TYPE csp_case_transport_status_enum :
(
	CSP_CASE_TRANSPORT_STATUS_NOT_INITIALIZED 							:=  0,
	CSP_CASE_TRANSPORT_STATUS_DISABLED 									:=  10,
	CSP_CASE_TRANSPORT_STATUS_ENABLE_REQUEST 							:=  20,
	CSP_CASE_TRANSPORT_STATUS_ENABLING 									:=  30,
	CSP_CASE_TRANSPORT_STATUS_ENABLED 									:=  40,
	CSP_CASE_TRANSPORT_STATUS_CHANGE_OVER_MODE							:=  45,
	CSP_CASE_TRANSPORT_STATUS_HOME_REQUEST								:=  50,
	CSP_CASE_TRANSPORT_STATUS_HOMING									:=  60,
	CSP_CASE_TRANSPORT_STATUS_HOME_DONE									:=  70,
	CSP_CASE_TRANSPORT_STATUS_CALCULATING_SLAVE_POSITION				:=  90,
	CSP_CASE_TRANSPORT_STATUS_CALCULATING_MASTER_POSITION				:=  91,
	CSP_CASE_TRANSPORT_STATUS_WAITING_SLAVE_ENGAGE						:= 100,
	CSP_CASE_TRANSPORT_STATUS_WAITING_MASTER_ENGAGE						:= 101,
	CSP_CASE_TRANSPORT_STATUS_PHASE_REQUEST								:= 140,
	CSP_CASE_TRANSPORT_STATUS_PHASING									:= 150,
	CSP_CASE_TRANSPORT_STATUS_PHASED									:= 160,
	CSP_CASE_TRANSPORT_STATUS_CAM_ENGAGED_REQ							:= 170,
	CSP_CASE_TRANSPORT_STATUS_AXIS_ENGAGE_VERIFY						:= 180,
	CSP_CASE_TRANSPORT_STATUS_CAM_ENGAGED								:= 190,
	CSP_CASE_TRANSPORT_STATUS_CAM_TABLE_READ							:= 195,
	CSP_CASE_TRANSPORT_STATUS_CALCULATE_SLAVE_POSITION_REQUEST			:= 196,
	CSP_CASE_TRANSPORT_STATUS_READY										:= 197,
	CSP_CASE_TRANSPORT_STATUS_RUNNING									:= 200,
	CSP_CASE_TRANSPORT_STATUS_MOVING									:= 205,
	CSP_CASE_TRANSPORT_STATUS_DISENGAGE_REQUEST							:= 210,
	CSP_CASE_TRANSPORT_STATUS_DISENGAGING								:= 211,	
	CSP_CASE_TRANSPORT_STATUS_STOP_REQUEST 								:= 500,
	CSP_CASE_TRANSPORT_STATUS_DISABLE_REQUEST 							:= 530,
	CSP_CASE_TRANSPORT_STATUS_DISABLING 								:= 540,
	
	CSP_CASE_TRANSPORT_STATUS_RECOVERY_CAM_ENGAGED_REQ					:= 305,
	CSP_CASE_TRANSPORT_STATUS_DISENGAGE_REJECT							:= 300,
	CSP_CASE_TRANSPORT_STATUS_REJECT_ABS_STEP_1							:= 301,
	CSP_CASE_TRANSPORT_STATUS_REJECT_ABS_STEP_2							:= 302,
	CSP_CASE_TRANSPORT_STATUS_REJECT_ABS_STEP_3							:= 303,
	CSP_CASE_TRANSPORT_STATUS_REJECT_ABS_STEP_4							:= 304	
	
) := CSP_CASE_TRANSPORT_STATUS_NOT_INITIALIZED;
END_TYPE

(* stored: Version 1.1.0.1, ProductVersion 3.1.4024.3
   DUT csp_case_transport_status_enum: Id {16332b9d-917f-46ac-ab8b-9641332c4766} *)
